FUNCTION TryConvert_DWORD_TO_BYTE : BOOL
VAR_INPUT
	in : DWORD;
	out : REFERENCE TO BYTE;
END_VAR

IF in > DatatypeLimits.MAX_VALUE_OF_DWORD_WHICH_CAN_BE_HELD_IN_A_BYTE THEN
	RETURN;
END_IF

out := DWORD_TO_BYTE(in);
TryConvert_DWORD_TO_BYTE := TRUE;

END_FUNCTION

(* stored: Version 1.1.0.1, ProductVersion 3.1.4024.12
   POU TryConvert_DWORD_TO_BYTE: Id {0823cb65-4f10-4bf3-8856-45bcddbaf64c}, SpecialFunc None *)
